KUKA KRL data list: ConfGarra_Wait.dat

&ACCESS RVO1
&REL 1
&PARAM EDITMASK = *
DEFDAT ConfGarra_Wait

ENDDAT
